// TIA Portal V19 export
TYPE "LEXCHANGETRAY_typePc_Status"
// stored: Access Published
   STRUCT
      Done : Bool;   // done
      error : Bool;   // error
      execute : Bool;   // execute
   END_STRUCT;
END_TYPE
